Staubli VAL3: onF4Event.pgx

program onF4Event()
  local num i
  local string l_sMessage
  local string l_sItem
begin
  // look if the bButton is enable
call loadPage("instrSequential/AXIS8/page_axis",l_sItem)
end
